FUNCTION_BLOCK FB_HeatExchanger1System EXTENDS FB_SystemContinous
VAR_INPUT
END_VAR
VAR_OUTPUT
END_VAR
VAR
	//default parameters
	localDefaultParameters : ST_HeatExchanger1DefaultParameters;

	//pumps
	stPU315DefaultParameters : ST_PumpGrundfosMagna3DefaultParameters := (tTaskCycleTime := GlobalVariables.tTaskCycleTime_MAIN, tCtrlCycleTime := GlobalVariables.tCtrlCycleTime_MAIN);
	stPU215DefaultParameters : ST_PumpGrundfosMagna3DefaultParameters := (bPumpBeforeApplication := FALSE, tTaskCycleTime := GlobalVariables.tTaskCycleTime_MAIN, tCtrlCycleTime := GlobalVariables.tCtrlCycleTime_MAIN);
	PU315 : FB_PumpGrundfosMagna3 := (ST_DefaultParameters := stPU315DefaultParameters);; 
	PU215 : FB_PumpGrundfosMagna3 := (ST_DefaultParameters := stPU215DefaultParameters);;

	//valves
	stSV315DefaultParameters : ST_DiscreteValveDefaultParameters := (nFeedback := 0);
	stRV215DefaultParameters : ST_MixingValveDefaultParameters := (bFeedbackSignal := TRUE, tTaskCycleTime := GlobalVariables.tCtrlCycleTime_MAIN, tCtrlCycleTime := GlobalVariables.tCtrlCycleTime_MAIN);
	
	SV315 : FB_DiscreteValve := (ST_DefaultParameters := stSV315DefaultParameters);
	RV215 : FB_MixingValve := (ST_DefaultParameters := stRV215DefaultParameters);
	
	//sensors
	WMZ215 : FB_MollineC3HeatCounter;
	
	//internal variables
	bSetStatusOn_PU315 : BOOL;
	bSetStatusOn_PU215 : BOOL;
	bSetStatusOn_SV315 : BOOL;
	bSetStatusOn_RV215 : BOOL;
	
	bStartTimer : BOOL;
	Timer : TON;
END_VAR

Timer(IN := bStartTimer,
	PT := T#75S);
MAIN();

//pumps
PU315.GetState_Profibus();
PU315(bSetStatusOnAutomatic := bSetStatusOn_PU315,
	fSetPointAutomatic := 70,
	bAlgorithmPermission := bAlgorithmPermission,
	nControlModeAutomatic := 1);
PU315.SetState_Profibus();

PU215.GetState_Profibus();
PU215(bSetStatusOnAutomatic := bSetStatusOn_PU215,
	fSetPointAutomatic := 70,
	bAlgorithmPermission := bAlgorithmPermission,
	nControlModeAutomatic := 0);
PU215.SetState_Profibus();

//valves
SV315.GetState_BI();
SV315(bSetStatusOnAutomatic := bSetStatusOn_SV315,
	bAlgorithmPermission := bAlgorithmPermission);
SV315.SetState_BO();

RV215.GetState_AI();
RV215(bSetStatusOnAutomatic := bSetStatusOn_RV215,
	fSetPointAutomatic := fSetPoint,
	bAlgorithmPermission := bAlgorithmPermission,
	fTemperatureExternal := PU215.fTemperatureInternal,
	nControlModeAutomatic := 2);
RV215.SetState_AO();

WMZ215(aHeatCounterTelegramm := Telegramm_WZ_PWT_1);

METHOD PROTECTED  CheckError : BOOL
VAR_INPUT
END_VAR
VAR_OUTPUT
	bError : BOOL;
END_VAR
bError := PU315.bError;
END_METHOD

METHOD PROTECTED  Operational : BOOL
VAR_INPUT
END_VAR
VAR_OUTPUT
	bSwitchToWorking : BOOL := FALSE;
END_VAR
bSetStatusOn_PU315 := TRUE;
bSetStatusOn_PU215 := TRUE;

IF PU315.bStatusOn AND PU215.bStatusOn THEN
	bSwitchToWorking := TRUE;
END_IF
END_METHOD

METHOD PROTECTED  RampDown : BOOL
VAR_INPUT
END_VAR
VAR_OUTPUT
	bRampDownFinished : BOOL := FALSE;
END_VAR
bSetStatusOn_PU215 := FALSE;
bSetStatusOn_PU315 := FALSE;

IF NOT PU315.bStatusOn AND NOT PU215.bStatusOn THEN
	bSetStatusOn_RV215 := FALSE;
	bSetStatusOn_SV315 := FALSE;
	bStartTimer := TRUE;
	IF Timer.Q AND RV215.fOperatingPoint<10 THEN
		bRampDownFinished := TRUE;
		bStartTimer := FALSE;
	END_IF
END_IF
END_METHOD

METHOD PROTECTED  RampUp : BOOL
VAR_INPUT
END_VAR
VAR_OUTPUT
	bRampUpFinished : BOOL := FALSE;
END_VAR
bSetStatusOn_SV315 := TRUE;
bSetStatusOn_RV215 := TRUE;

bStartTimer := TRUE;
IF Timer.Q THEN
	bStartTimer := FALSE;
	bRampUpFinished := TRUE;
END_IF
END_METHOD

METHOD PROTECTED   SetSetPointLimits : BOOL
VAR_INPUT
END_VAR
aSetPointLimits[1] := localDefaultParameters.aSetPointLimitsTemperature[1];
aSetPointLimits[2] := localDefaultParameters.aSetPointLimitsTemperature[2];
END_METHOD

METHOD PROTECTED  SetState : BOOL
VAR_INPUT
END_VAR
VAR_OUTPUT
END_VAR
fOperatingPoint := PU215.fTemperatureInternal;

controlState.bStatusOn := bSetStatusOn;
setPointState.aSetPointLimits := aSetPointLimits;
setPointState.fSetPoint := fSetPoint;
setPointState.fOperatingPoint := fOperatingPoint;
setPointState.sSetPointUnit := 'degreeC';
setPointState.sOperatingPointUnit := 'degreeC';
END_METHOD

METHOD PROTECTED  Working : BOOL
VAR_INPUT
END_VAR
VAR_OUTPUT
	bSwitchToOperational : BOOL := FALSE;
END_VAR
//empty method
END_METHOD

END_FUNCTION_BLOCK

(* stored: Version 1.1.0.1, ProductVersion 3.1.4024.10
   POU FB_HeatExchanger1System: Id {bca56c6b-1b09-4f57-a186-5b7562770c5b}, SpecialFunc None
   Method CheckError: Id {b54ba0ca-5b25-4c17-92f0-eb09cfdea800}
   Method Operational: Id {7ac6e3b2-880f-4ae7-8766-d8b22693c3d9}
   Method RampDown: Id {38be2d03-34bf-4165-98f1-2ff7a50120b6}
   Method RampUp: Id {79fc56b0-c2f3-4502-acb0-473bf863e404}
   Method SetSetPointLimits: Id {08b841e3-f57f-4525-b475-9463ff8dff61}
   Method SetState: Id {9b468ecf-33a9-49ee-a2cd-1270fe631d8f}
   Method Working: Id {2d7be513-42f4-4f0a-9e3f-306a74f1d37d} *)
